(* PLC project Unnamed, Unknown Unnamed 1 *)
(* stored: creationDateTime 2020-11-16T20:33:12, modificationDateTime 2020-11-16T20:33:12 *)

CONFIGURATION Config0
  RESOURCE Res0 ON PLC
  END_RESOURCE
END_CONFIGURATION
